// TIA Portal V21 export
FUNCTION "fcSafety" : Void   // FC1, LAD
{ S7_Optimized_Access := 'TRUE' }
// stored: SetENOAutomatically false
BEGIN

REGION Network 1: Safety
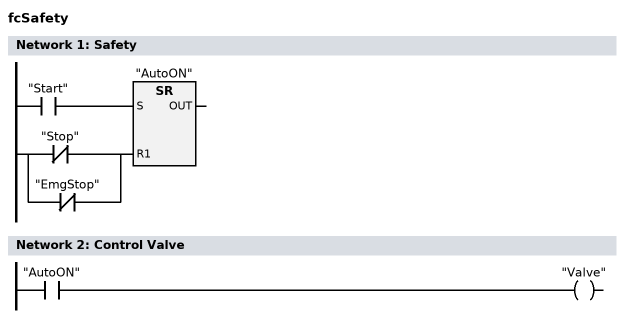
   RUNG wire#powerrail
      Contact( "Start" )
      S_SR(operand := "AutoON", r1 := wire#w1)
   END_RUNG
   RUNG wire#powerrail
      I_Contact( "Stop" )
   END_RUNG wire#w1
   RUNG wire#powerrail
      I_Contact( "EmgStop" )
   END_RUNG wire#w1
   // the same network as SCL:
   IF "Start" THEN
       "AutoON" := TRUE;   // SR flip-flop
   END_IF;
   IF NOT "Stop" OR NOT "EmgStop" THEN "AutoON" := FALSE; END_IF;
END_REGION

REGION Network 2: Control Valve
   RUNG wire#powerrail
      Contact( "AutoON" )
      Coil( "Valve" )
   END_RUNG
   // the same network as SCL:
   "Valve" := "AutoON";
END_REGION
END_FUNCTION
